FUNCTION_BLOCK FB_EndlessExtruderTMCM_Ref EXTENDS FB_ExtruderRef
VAR_INPUT
END_VAR
VAR
	pHwRefTMCM1140 	: POINTER TO FB_HwRefTMCM1140;
	eTriggerOutput	: E_TriggerOutput;
	nTriggerChannel	: USINT;	
END_VAR
VAR_OUTPUT
END_VAR

METHOD FB_init : BOOL
VAR_INPUT
	bInitRetains 	: BOOL; // if TRUE, the retain variables are initialized (warm start / cold start)
	bInCopyCode 	: BOOL;  // if TRUE, the instance afterwards gets moved into the copy code (online change)
	pHwRefTMCM1140 	: POINTER TO FB_HwRefTMCM1140;
	//eTriggerOutput	: E_TriggerOutput;
	//nTriggerChannel	: USINT;
END_VAR
THIS^.pHwRefTMCM1140 := pHwRefTMCM1140;
//THIS^.eTriggerOutput := eTriggerOutput;
//THIS^.nTriggerChannel := nTriggerChannel;
END_METHOD

PROPERTY P_bError : BOOL
GET
END_GET
END_PROPERTY

PROPERTY P_bIsActive : BOOL
GET
END_GET
END_PROPERTY

PROPERTY P_bIsLocked : BOOL
GET
P_bIsLocked := TRUE;
END_GET
END_PROPERTY

PROPERTY P_eTriggerOutput : E_TriggerOutput
GET
P_eTriggerOutput := eTriggerOutput;
END_GET
END_PROPERTY

PROPERTY P_nTriggerChannel : USINT
GET
P_nTriggerChannel := nTriggerChannel;
END_GET
END_PROPERTY

PROPERTY P_pHwRefTMCM1140 : POINTER TO FB_HwRefTMCM1140
GET
P_pHwRefTMCM1140 := pHwRefTMCM1140;
END_GET
END_PROPERTY

END_FUNCTION_BLOCK

(* stored: Version 1.1.0.1, ProductVersion 3.1.4024.11
   POU FB_EndlessExtruderTMCM_Ref: Id {7295e60e-54b6-4fec-85c4-5c7e28d7ec40}, SpecialFunc None
   Method FB_init: Id {a8ae3470-e4bf-403a-9f75-c3ef8fbeb2bc}
   Property P_bError: Id {17a7ec3e-2970-483d-97a8-a2c4452afadf}
   Get Get: Id {9e961f29-d2b6-47bf-89e2-9455c3c8160e}
   Property P_bIsActive: Id {840c16fa-c4bd-4e8e-ae7b-8e86bddb17b8}
   Get Get: Id {cebe5ff6-a67f-4eed-8d8b-08ad259440f8}
   Property P_bIsLocked: Id {f67ba6a1-ddfb-4f90-ad6c-08f467464dfb}
   Get Get: Id {e2802494-1fc0-4882-b46d-fdfa69fc691d}
   Property P_eTriggerOutput: Id {6a3263d0-eaf8-4701-8cb6-33669840ab00}
   Get Get: Id {7fc66a21-02a1-4dac-83d3-498502d450ad}
   Property P_nTriggerChannel: Id {ed2eed39-265a-4ef0-8e24-6d43b8bbee1e}
   Get Get: Id {78515e3b-f0c7-4fba-9723-c2de4087d385}
   Property P_pHwRefTMCM1140: Id {d421782e-1f55-42de-9c30-62d838764e54}
   Get Get: Id {704de267-9e18-499f-8a04-9de68f37d650} *)
